SUBAPPLICATION Uebung_010b5 (* SoftKey_F1-10 auf DigitalOutput_Q1-10 *)
  (* Standard: 61499-2; Description: Copyright (c) 2023 Meisterschulen am Ostbahnhof This program and the accompanying materials are made available under the terms of the Eclipse Public License 2.0 which is available at https://www.eclipse.org/legal/epl-2.0/ SPDX-License-Identifier: EPL-2.0 *)
  (* Version 1.0, 2023-10-23, Franz Höpfinger, Meisterschulen am Ostbahnhof *)
  PACKAGE Uebungen;
  IMPORT Uebungen::const::UT::DefaultPool::SoftKey_F1;
  IMPORT Uebungen::const::UT::DefaultPool::SoftKey_F10;
  IMPORT Uebungen::const::UT::DefaultPool::SoftKey_F2;
  IMPORT Uebungen::const::UT::DefaultPool::SoftKey_F3;
  IMPORT Uebungen::const::UT::DefaultPool::SoftKey_F4;
  IMPORT Uebungen::const::UT::DefaultPool::SoftKey_F5;
  IMPORT Uebungen::const::UT::DefaultPool::SoftKey_F6;
  IMPORT Uebungen::const::UT::DefaultPool::SoftKey_F7;
  IMPORT Uebungen::const::UT::DefaultPool::SoftKey_F8;
  IMPORT Uebungen::const::UT::DefaultPool::SoftKey_F9;
  IMPORT logiBUS::io::DQ::logiBUS_DO::Output_Q1;
  IMPORT logiBUS::io::DQ::logiBUS_DO::Output_Q10;
  IMPORT logiBUS::io::DQ::logiBUS_DO::Output_Q2;
  IMPORT logiBUS::io::DQ::logiBUS_DO::Output_Q3;
  IMPORT logiBUS::io::DQ::logiBUS_DO::Output_Q4;
  IMPORT logiBUS::io::DQ::logiBUS_DO::Output_Q5;
  IMPORT logiBUS::io::DQ::logiBUS_DO::Output_Q6;
  IMPORT logiBUS::io::DQ::logiBUS_DO::Output_Q7;
  IMPORT logiBUS::io::DQ::logiBUS_DO::Output_Q8;
  IMPORT logiBUS::io::DQ::logiBUS_DO::Output_Q9;
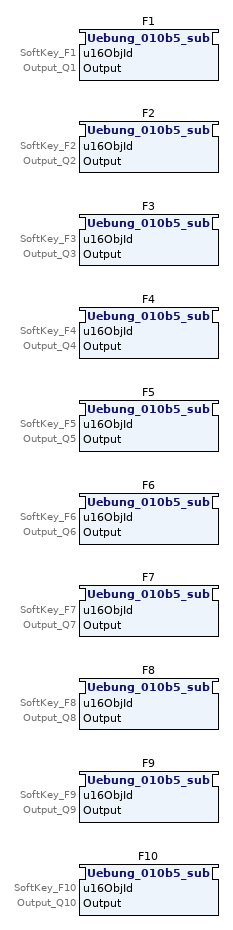
  SUBAPPS
    F1 : Uebungen::Uebung_010b5_sub(u16ObjId := SoftKey_F1, Output := Output_Q1);
    F2 : Uebungen::Uebung_010b5_sub(u16ObjId := SoftKey_F2, Output := Output_Q2);
    F3 : Uebungen::Uebung_010b5_sub(u16ObjId := SoftKey_F3, Output := Output_Q3);
    F4 : Uebungen::Uebung_010b5_sub(u16ObjId := SoftKey_F4, Output := Output_Q4);
    F5 : Uebungen::Uebung_010b5_sub(u16ObjId := SoftKey_F5, Output := Output_Q5);
    F6 : Uebungen::Uebung_010b5_sub(u16ObjId := SoftKey_F6, Output := Output_Q6);
    F7 : Uebungen::Uebung_010b5_sub(u16ObjId := SoftKey_F7, Output := Output_Q7);
    F8 : Uebungen::Uebung_010b5_sub(u16ObjId := SoftKey_F8, Output := Output_Q8);
    F9 : Uebungen::Uebung_010b5_sub(u16ObjId := SoftKey_F9, Output := Output_Q9);
    F10 : Uebungen::Uebung_010b5_sub(u16ObjId := SoftKey_F10, Output := Output_Q10);
  END_SUBAPPS
END_SUBAPPLICATION
